{attribute 'GeneratedUsingTerminal: EL3204-0200-0016'}
{attribute addProperty BoxType "EL3204-0200-0016"}
{attribute addProperty Id "RTD_Inputs_Channel_1AT %I*RTD_Inputs_Channel_9575FEA17RTD_Inputs_Channel_2AT %I*RTD_Inputs_Channel_9575FEA17RTD_Inputs_Channel_3AT %I*RTD_Inputs_Channel_9575FEA17RTD_Inputs_Channel_4AT %I*RTD_Inputs_Channel_9575FEA17WcStateAT %I*WcState_9091E0EB2InfoDataAT %I*InfoData_94A18F5E2"}
{attribute addProperty CRC "1709700539"}
{attribute addProperty Size "32"}
TYPE EL3204_65E7F5BB EXTENDS EtcSlaveTerminalBase_947E5A46 :
STRUCT
	{attribute addProperty Name "RTD_Inputs_Channel_1"}
	RTD_Inputs_Channel_1 : RTD_Inputs_Channel_9575FEA1;
	{attribute addProperty Name "RTD_Inputs_Channel_2"}
	RTD_Inputs_Channel_2 : RTD_Inputs_Channel_9575FEA1;
	{attribute addProperty Name "RTD_Inputs_Channel_3"}
	RTD_Inputs_Channel_3 : RTD_Inputs_Channel_9575FEA1;
	{attribute addProperty Name "RTD_Inputs_Channel_4"}
	RTD_Inputs_Channel_4 : RTD_Inputs_Channel_9575FEA1;
	{attribute addProperty Name "WcState"}
	WcState : WcState_9091E0EB;
	{attribute addProperty Name "InfoData"}
	InfoData : InfoData_94A18F5E;
END_STRUCT
END_TYPE

(* stored: Version 1.2.0.0, ProductVersion 3.1.4024.9
   DUT EL3204_65E7F5BB: Id {158cea09-0110-476c-bf2f-81afe55b01a7} *)
